RoboDK station: PyndoBots.rdk

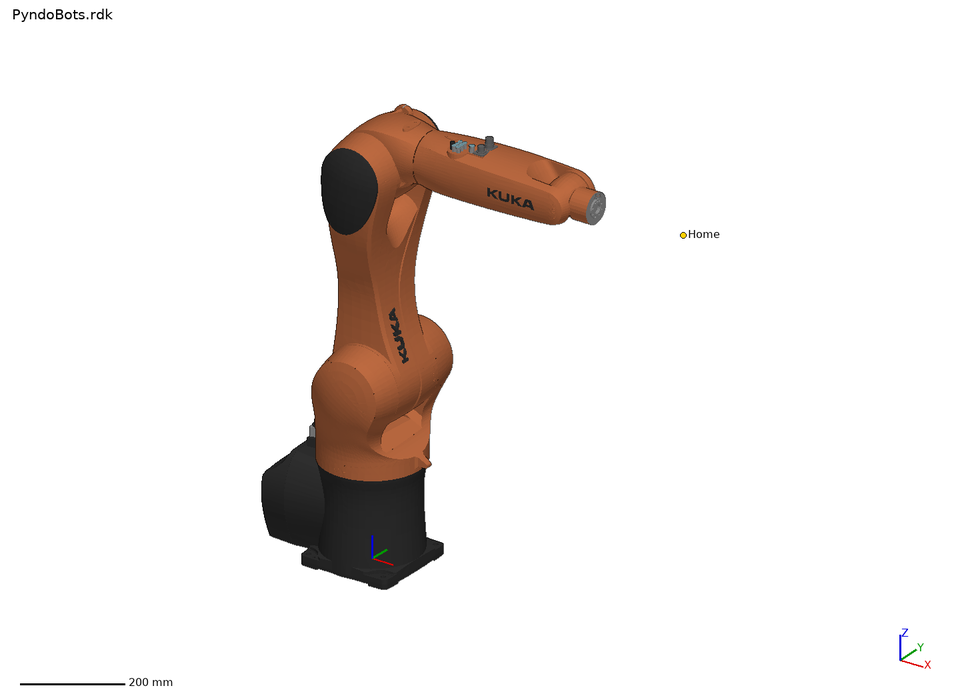
[picture v0: the station drawn from its stored meshes, robots at their saved joint values, targets as dots, program paths as lines]
Station PyndoBots (saved by RoboDK 5.2.1). Poses are relative to the parent item; angles as X-Y-Z fixed-axis rotations.
  - frame KUKA KR 6 R900 sixx Base at (0, 0, 0) mm
    - robot KUKA KR 6 R900 sixx: 6 axes, payload 6 kg, reach 901 mm, repeatability 0.03 mm, weight 52 kg
        modified DH rows (alpha deg, a mm, theta deg, d mm): 0, 0, 0, 400; -90, 25, 0, 0; 0, 455, -90, 0; -90, 35, 0, 420; 90, 0, 0, 0; -90, 0, 180, 80
        joint limits [-170, -190, -120, -185, -120, -350] to [170, 45, 156, 185, 120, 350]; home [0, -90, 90, 0, 0, 0]; saved at [0, -90, 90, 0, 0, 0]
      - tool Weild Gun, TCP at (0, 0, 200) mm
    - target Home (Cartesian target) at (725, 0, 890) mm, rotated rx 0 ry 90 rz 0 deg; joints [0, -90, 90, 0, 0, 0] of KUKA KR 6 R900 sixx
    - target Target 1 (Cartesian target) at (725, 0, 890) mm, rotated rx 0 ry 90 rz 0 deg; joints [0, -90, 90, 0, 0, 0] of KUKA KR 6 R900 sixx
  - Python program PyndoBot (listed below)

--- Python program PyndoBot ---

